// Interlocks share data for synced operation with other blocks
INTERFACE I_MotionInterlocksShareData

PROPERTY AxisError : BOOL
GET
END_GET
END_PROPERTY

PROPERTY BrakeError : BOOL
GET
END_GET
END_PROPERTY

PROPERTY GlobalReset : BOOL
GET
END_GET
END_PROPERTY

PROPERTY HomeBusy : BOOL
GET
END_GET
END_PROPERTY

PROPERTY LimBackward : BOOL
GET
END_GET
END_PROPERTY

PROPERTY LimForward : BOOL
GET
END_GET
END_PROPERTY

PROPERTY LimHome : BOOL
GET
END_GET
END_PROPERTY

PROPERTY MoveDone : BOOL
GET
END_GET
END_PROPERTY

END_INTERFACE

(* stored: Version 1.1.0.1
   Itf I_MotionInterlocksShareData: Id {f664124a-a4eb-460c-beeb-498daf79d1c6}
   Property AxisError: Id {791a0996-afd2-49f3-b52f-3cbd46ef51c9}
   Get Get: Id {2aa30525-6630-4d08-bd1f-c5fd1296dbb1}
   Property BrakeError: Id {33aedee8-8240-4128-929f-9b1eed4d89e5}
   Get Get: Id {bc630ab7-e97e-4fb1-b9ab-c242b0c547b1}
   Property GlobalReset: Id {3cb9be1b-8a2f-4d9a-aeed-5fa8a8a4a1f3}
   Get Get: Id {cbce352f-7209-4323-97a9-2a34ea09e939}
   Property HomeBusy: Id {2382ab9e-e464-498b-b3d1-3eb574860f78}
   Get Get: Id {35889636-b658-4fba-89f2-a1033924d466}
   Property LimBackward: Id {be547acb-e1fd-4050-bb2d-6f025603040d}
   Get Get: Id {cbdd562a-99aa-4b0f-97bd-ef35d7db9102}
   Property LimForward: Id {507a6415-3928-42e3-8134-3e476dbbb9d5}
   Get Get: Id {2453c3d3-ce7e-4ff9-94f7-452773acc1fb}
   Property LimHome: Id {7438c6e7-800b-414c-9ad6-226a2391d055}
   Get Get: Id {7a8a0145-1223-4fa8-a7c1-ebe32e3b2b81}
   Property MoveDone: Id {5e0e073b-50c5-4948-be6f-702b298fdd9b}
   Get Get: Id {f6af31e0-cb12-4de7-b30f-e64dd9ed7440} *)
